{attribute addProperty BoxType "EL2794-0000-0016"}
{attribute addProperty Id "ChannelAT %Q*ARRAY[0..3] OF Channel_7F374EB03240WcStateAT %I*WcState_64F6A8C6810InfoDataAT %I*InfoData_192954DE1620"}
{attribute addProperty CRC "999552494"}
{attribute addProperty SizeInBites "56"}
{attribute addProperty SizeInBytes "7"}
TYPE EL2794_E7E37CC2 :
STRUCT
	{attribute addProperty Name "Channel"}
	Channel : ARRAY[0..3] OF Channel_7F374EB0;
	{attribute addProperty Name "WcState"}
	WcState : WcState_64F6A8C6;
	{attribute addProperty Name "InfoData"}
	InfoData : InfoData_192954DE;
END_STRUCT
END_TYPE

(* stored: Version 1.2.0.0, ProductVersion 3.1.4024.9
   DUT EL2794_E7E37CC2: Id {6b802219-eb80-49ec-9c65-e34787e956b6} *)
